RoboDK station: RoboDK sw03 Station UR3e mit Gripper.rdk

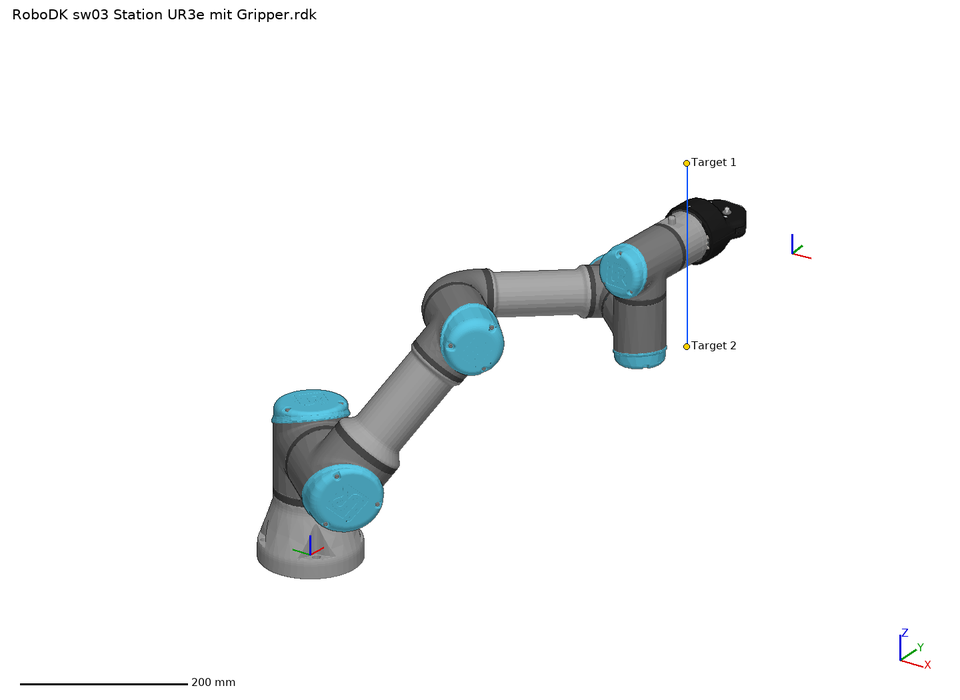
[picture v0: the station drawn from its stored meshes, robots at their saved joint values, targets as dots, program paths as lines]
Station UR3e_Station_SRO01 (saved by RoboDK 5.9.5). Poses are relative to the parent item; angles as X-Y-Z fixed-axis rotations.
Station parameters (name, value as stored): OPC-UA, opc.tcp://localhost:4840
  - frame UR3e Base at (0, 0, 0) mm, rotated rx 0 ry 0 rz 87.34 deg
    - robot UR3e: 6 axes, payload 3 kg, reach 500 mm, repeatability 0.03 mm, weight 11 kg
        modified DH rows (alpha deg, a mm, theta deg, d mm): 0, 0, 0, 151.9; 90, 0, 180, 0; 0, 243.55, 0, 0; 0, 213.2, 0, 131.05; -90, 0, 0, 85.35; 90, 0, 180, 92.1
        joint limits [-360, -360, -360, -360, -360, -360] to [360, 360, 360, 360, 360, 360]; home [0, -90, -90, 0, 90, 0]; saved at [-37.75, -130.655, -54.204, 4.859, 127.75, 0]
      - robot RobotiQ 2F85: 1 axes, payload 5 kg
          joint limits [0] to [85]; home [85]; saved at [85]
    - target Target 1 (Cartesian target) at (305.3, -330.82, 499.85) mm, rotated rx -90 ry 0 rz -90 deg; joints [-37.75, -139.539, -11.094, -29.367, 127.75, 0] of UR3e
    - target Target 2 (Cartesian target) at (305.3, -330.82, 257.13) mm, rotated rx -90 ry 0 rz -90 deg; joints [-37.75, -144.026, -71.271, 35.297, 127.75, 0] of UR3e
  - frame RobotiQ 2F85 Base at (0, 1000, 0) mm, rotated rx 0 ry 0 rz 6.01 deg
  - program Prog1 (5 instructions, listed below)

--- program Prog1 (robot UR3e) ---
  Set Ref.: UR3e Base
  MoveJ (Target 1)
  Pause 500 ms
  MoveL (Target 2)
  Pause 500 ms
